TYPE ST_RecipeList :
STRUCT
	sName			:STRING;
	sCreated		:STRING;
	sEdited			:STRING;
	sVerified		:STRING[3];
END_STRUCT
END_TYPE

(* stored: Version 1.1.0.1, ProductVersion 3.1.4024.12
   DUT ST_RecipeList: Id {3aacd1e5-e1a4-4705-9460-b12856c1969f} *)
